# EPICS substitutions: src/main/epics/wtrvac-freiaApp/Db/vac.substitutions
file "TP_AI.template" { pattern
{P,  		    SIG,	OFFS, TYP,    PREC,   EGU,   LOPR,  HOPR, H,	MAXVAL, PB_ADDR}
{CstatH-Vac:TP001,   MotV,	248,  BYTE,   0,      "V",   0,	100,	100,	100,	5}
{CstatH-Vac:TP001,   BearingT,	249,  BYTE,   0,      "°C",  0,	100,	100,	100,	5}
{CstatH-Vac:TP001,   PSupplyT,	250,  BYTE,   0,      "°C",  0,	100,	100,	100,	5}
{CstatH-Vac:TP001,   CPU_T,	251,  BYTE,   0,      "°C",  0,	100,	100,	100,	5}
{CstatH-Vac:TP001,   MotI,	256,  UINT16, 3,      "A",   0,	10,	10000,	10,	5}
{CstatH-Vac:TP001,   MotP,	258,  UINT16, 0,      "W",   0,	200,	200,	200,	5}
{CstatH-Vac:TP001,   MotPLimit,	260,  UINT16, 0,      "W",   0,	200,	200,	200,	5}
{CstatH-Vac:TP001,   Freq,	262,  UINT16, 0,      "Hz",  0,	1500,	1500,	1500,	5}
{CstatH-Vac:TP001,   FreqSP,	264,  UINT16, 0,      "Hz",  0,	1500,	1500,	1500,	5}
{CstatH-Vac:TP001,   NoOfStarts,266,  UINT16, 0,      "",    0,	65535,	65535,	65535,	5}
{CstatH-Vac:TP001,   LastOnTime,268,  UINT16, 0,      "min.",0,	65535,	65535,	65535,	5}
{CstatH-Vac:TP001,   OpTime,	270,  UINT16, 0,      "h",   0,	65535,	65535,	65535,	5}
{CstatH-Vac:TP002,   Freq,	278,  UINT16, 0,      "Hz",  0,	1000,	1000,	1000,	6}
{CstatV-Vac:TP050,   Freq,	742,  UINT16, 0,      "Hz",  0,	1000,	1000,	1000,	8}
{CstatV-Vac:TP060,   Freq,	906,  UINT16, 0,      "Hz",  0,	1000,	1000,	1000,	9}
}

file "CtrlBitwRdBack.template" { pattern

{P,                   SIG,	S_OFFS, S_BIT, S_ZNAM, S_ONAM, C_OFFS, C_BIT, C_ZNAM,   C_ONAM,	INIT_EVNT}
{CstatH-Vac:TP002,    Remote,	276,	 7     Local,  Remote, 46,	  2,	 Local, Remote,	7}
{CstatV-Vac:TP050,    Remote,	740,	 7     Local,  Remote, 144,	  2,	 Local, Remote,	7}
{CstatV-Vac:TP060,    Remote,	904,	 7     Local,  Remote, 194,	  2,	 Local, Remote,	7}
#{CstatH-Vac:TP002,    On,	276,	 2     OFF,    ON,     47,	  0,	 Stop,  Start,	7}
}
